(* PLC project Hello Mixing tank, CODESYS CODESYS V3.5 SP16, author Toni Kucic *)
(* stored: creationDateTime 2021-03-11T21:02:17.1386427, version 1.0, modificationDateTime 2021-03-11T20:32:57.2894189, organization Tk Automation *)
(* In industrial automation the "hello world" program is a mixing tank. As a part of my portfolio I have written a simple mixing tank controller and a simulator. The project is meant for begginers and for educational purposes. It is published under MIT license. Written in CODESYS 3.5 and in structured text language.

The project is designed in a way that the user can disable the main program and replace it with his own implementation. Simulator and the HMI sees only the IO and HMI global variables so if the user wishes to create an own implementation those variables should be written. On the simulator side the operator can see if the implementation is working correctly. *)

(* values of MODES: MANUAL: System is in manual mode (Operator control); AUTO: System is in auto mode (PLC in control) *)

{attribute 'qualified_only'}
{attribute 'strict'}
TYPE MODES : (MANUAL := 0, AUTO := 1);
END_TYPE

(* values of AUTO_SEQUENCE: DRAINING: Draining state when system is in auto mode; FILLING: Filling state when system is in auto mode; MIXING: Mixing state when system is in auto mode *)

{attribute 'qualified_only'}
{attribute 'strict'}
TYPE AUTO_SEQUENCE : (DRAINING := 0, FILLING := 1, MIXING := 2);
END_TYPE

FUNCTION_BLOCK GenericBistableDeviceModel
  VAR_INPUT
    ActivateCmd : BOOL;  (* Command to activate the device *)
    DeactivateCmd : BOOL;  (* Command to deactivate the device *)
    cfgActTime : TIME := TIME#1s0ms;  (* Time needed to activate the device *)
    cfgDeactTime : TIME := TIME#1s0ms;  (* Time needed to deactivate the device *)
    simActFail : BOOL;  (* Simulates activation fail. If deactivated and activate command true. *)
    simDeactFail : BOOL;  (* Simulates deactivation fail. If activated and deactivate command true. *)
  END_VAR
  VAR_OUTPUT
    Activated : BOOL;  (* TRUE: Device is activated *)
    Deactivated : BOOL;  (* TRUE: Device is deactivated *)
  END_VAR
  VAR
    TransitionDelay : TON;  (* Timer for delaying the commands to change state *)
    vState : USINT := 0;  (* State tracking variable *)
    vStateOld : USINT := 3;  (* Memory of previous state *)
  END_VAR

            CASE vState OF
	0: (*Deactivated*)
		(*On entry do:*)
		IF vState <> vStateOld THEN
			(*Reset timer*)
			TransitionDelay(IN:=FALSE);
			vStateOld := vState;
		END_IF
		TransitionDelay(IN:=ActivateCmd AND NOT simActFail, PT:=cfgActTime);
		IF TransitionDelay.Q THEN
			vState := 1;
		END_IF
	1: (*Activated*)
		(*On entry do:*)
		IF vState <> vStateOld THEN
			(*Reset timer*)
			TransitionDelay(IN:=FALSE);
			vStateOld := vState;
		END_IF
		TransitionDelay(IN:=DeactivateCmd AND NOT simDeactFail, PT:=cfgDeactTime);
		IF TransitionDelay.Q THEN
			vState := 0;
		END_IF
END_CASE
Activated := vState = 1;
Deactivated := vState = 0;
          
END_FUNCTION_BLOCK

PROGRAM simulator
  VAR
    vTankLevel : REAL := 25;  (* Simulated tank level, intialized to 25% *)
    MixerMotor : GenericBistableDeviceModel;  (* Simulated mixer motor *)
    MediumValve1 : GenericBistableDeviceModel;  (* Simulated valve that fills medium 1 *)
    MediumValve2 : GenericBistableDeviceModel;  (* Simulated valve that fills medium 2 *)
    DrainValve : GenericBistableDeviceModel;  (* Simulated valve that drains the tank *)
    vMotorRotating : REAL;  (* Motor activated for HMI *)
  END_VAR

                    (*Motor and valve simulation*)
MixerMotor(
	ActivateCmd := IO.xDO_M1_MixerMotorRunCmd,
	DeactivateCmd := NOT IO.xDO_M1_MixerMotorRunCmd,
	cfgActTime := T#2S,
	cfgDeactTime := T#0S,
	Activated => IO.xDI_M1_MixerMotorRunning);

MediumValve1(
	ActivateCmd := IO.xDO_VV01_Medium1_OpenCmd,
	DeactivateCmd := NOT IO.xDO_VV01_Medium1_OpenCmd,
	cfgActTime := T#1S,
	cfgDeactTime := T#1S,
	Activated => IO.xDI_VV01_Medium1_Opened);

MediumValve2(
	ActivateCmd := IO.xDO_VV02_Medium2_OpenCmd,
	DeactivateCmd := NOT IO.xDO_VV02_Medium2_OpenCmd,
	cfgActTime := T#1S,
	cfgDeactTime := T#1S,
	Activated => IO.xDI_VV02_Medium2_Opened);

DrainValve(
	ActivateCmd := IO.xDO_VV03_TankDrain_OpenCmd,
	DeactivateCmd := NOT IO.xDO_VV03_TankDrain_OpenCmd,
	cfgActTime := T#1S,
	cfgDeactTime := T#1S,
	Activated => IO.xDI_VV03_TankDrain_Opened);
	
(*Tank filling simulation*)
(*Tank fills if either filling valves are open and drains if the drain is open,
if the program overfills it, the tank spills to the spill way*)
vTankLevel :=  vTankLevel
			 + 0.1 * BOOL_TO_REAL(MediumValve1.Activated)
			 + 0.1 * BOOL_TO_REAL(MediumValve2.Activated)
			 - 0.2 * BOOL_TO_REAL(DrainValve.Activated);
vTankLevel := LIMIT(0, vTankLevel, 100);

(*Limit switch simulation*)
IO.xDI_LS01_TankLevelFull := vTankLevel >= 85;
IO.xDI_LS02_TankLevelEmpty := vTankLevel <= 5;

(*HMI *)
vMotorRotating := vMotorRotating + 1 * BOOL_TO_REAL(MixerMotor.Activated);
IF vMotorRotating >= 360 THEN vMotorRotating := 0; END_IF

                  
END_PROGRAM

PROGRAM main
  VAR
    vMode : MODES;  (* Variable to keep track of system mode Manual/Auto *)
    vModeOld : MODES;  (* Memory of last mode *)
    vAutoState : AUTO_SEQUENCE;  (* Variable to track the automatic sequence *)
    MixingTimer : TON;  (* Timer to control the mixing duration *)
  END_VAR

                    (*Functional description:
There are two ways of operation:
	- Manual
	- Automatic
Manual:
	- Operator is able to operate each valve manually
	- Operator is able to operate the mixer motor manually
	- Overfill protections are disabled
	- Operator is able to put the system to auto
	
Automatic:
	- Program will automatically control the valves and the mixing motor if system is in auto
	- If the tanks level is undefined it assumes draining state
	- In draining state, drains the tank until LS02 activates (tank is empty)
	- When tank is empty, it activates the medium 1 and 2 valves, closes the drain valve and the tank is filling up
	- Filling state is until LS01 is activated (Tank is full)
	- Then the mixer motor is mixing for 10 seconds
	- After mixing is completed, drain the whole contents
	- Repeats as long as auto is activated
	
HMI Requirements:
	- Manual / Auto needs to be correctly controlled and displayed
	- If manual, clicking on devices activates or stops them
	- If auto, clicking is not doing anything
	- If auto, system is counting number of cycles completed
	- Devices must clearly display if they are activated or deactivated*)

(*Enabling operator to select auto or manual mode*)
CASE vMode OF
	MODES.AUTO:
		IF HMI.SetToManual THEN
			vMode := Modes.MANUAL;
			HMI.SetToManual := FALSE;
		END_IF
		
	MODES.MANUAL:
		IF HMI.SetToAuto THEN
			vMode := Modes.AUTO;
			HMI.SetToAuto := FALSE;
		END_IF
END_CASE

(*Control of the system*)
CASE vMode OF
	MODES.MANUAL: (*Manual*)
		(*On entry do:*)
		IF vMode <> vModeOld THEN
			vAutoState := AUTO_SEQUENCE.DRAINING;
			vModeOld := vMode;
		END_IF
		
		(*In manual, HMI commands are connected to the IO for starting and stopping the devices*)
		(*Commands are implemented with a latch*)
		IO.xDO_M1_MixerMotorRunCmd := (HMI.MixerRunCmd OR IO.xDI_M1_MixerMotorRunning) AND NOT (HMI.MixerStopCmd);
		IO.xDO_VV01_Medium1_OpenCmd := (HMI.Medium1OpenCmd OR IO.xDI_VV01_Medium1_Opened) AND NOT (HMI.Medium1CloseCmd);
		IO.xDO_VV02_Medium2_OpenCmd := (HMI.Medium2OpenCmd OR IO.xDI_VV02_Medium2_Opened) AND NOT (HMI.Medium2CloseCmd);
		IO.xDO_VV03_TankDrain_OpenCmd := (HMI.DrainOpenCmd OR IO.xDI_VV03_TankDrain_Opened) AND NOT (HMI.DrainCloseCmd);
	
	MODES.AUTO: (*Automatic*)
		(*On entry do:*)
		IF vMode <> vModeOld THEN
			vAutoState := AUTO_SEQUENCE.DRAINING;
			vModeOld := vMode;
		END_IF
		CASE vAutoState OF
			AUTO_SEQUENCE.FILLING:
				(*Make sure other devices are not working*)
				IO.xDO_M1_MixerMotorRunCmd := FALSE;
				IO.xDO_VV03_TankDrain_OpenCmd := FALSE;
				
				(*Open both medium valves and start filling the tank*)
				IO.xDO_VV01_Medium1_OpenCmd := NOT IO.xDI_LS01_TankLevelFull;
				IO.xDO_VV02_Medium2_OpenCmd := NOT IO.xDI_LS01_TankLevelFull;
				
				(*When tank is full, wait for the filling valves to close and then go to mixing state*)
				IF IO.xDI_LS01_TankLevelFull AND NOT (IO.xDI_VV01_Medium1_Opened OR IO.xDI_VV02_Medium2_Opened) THEN
					vAutoState := AUTO_SEQUENCE.MIXING;
				END_IF
			AUTO_SEQUENCE.MIXING:
				(*Make sure other devices are not working*)
				IO.xDO_VV01_Medium1_OpenCmd := FALSE;
				IO.xDO_VV02_Medium2_OpenCmd := FALSE;
				IO.xDO_VV03_TankDrain_OpenCmd := FALSE;
				
				(*Start the mixer motor and mix for 10s*)
				IO.xDO_M1_MixerMotorRunCmd := TRUE;
				MixingTimer(IN:=IO.xDI_M1_MixerMotorRunning, PT:=T#10S);
				
				(*When timer has elapsed 10s, wait for motor to stop running, then go to draining*)
				IF MixingTimer.Q THEN
					IO.xDO_M1_MixerMotorRunCmd := FALSE;
					vAutoState := AUTO_SEQUENCE.DRAINING;
				END_IF
				
			AUTO_SEQUENCE.DRAINING:
				(*Make sure other devices are not working*)
				IO.xDO_M1_MixerMotorRunCmd := FALSE;
				IO.xDO_VV01_Medium1_OpenCmd := FALSE;
				IO.xDO_VV02_Medium2_OpenCmd := FALSE;
				
				(*Open the drain valve and start draining the tank*)
				IO.xDO_VV03_TankDrain_OpenCmd := NOT IO.xDI_LS02_TankLevelEmpty;
				
				(*When the tank is empty, wait for the drain valve to close,then go to filling*)
				IF IO.xDI_LS02_TankLevelEmpty AND NOT IO.xDI_VV03_TankDrain_Opened THEN
					vAutoState := AUTO_SEQUENCE.FILLING;
					HMI.CyclesCompleted := HMI.CyclesCompleted + 1;
				END_IF
		END_CASE
END_CASE

(*Command sanity reset*)
IF IO.xDI_M1_MixerMotorRunning THEN
	HMI.MixerRunCmd := FALSE;
ELSE
	HMI.MixerStopCmd := FALSE;
END_IF
IF IO.xDI_VV01_Medium1_Opened THEN
	HMI.Medium1OpenCmd := FALSE;
ELSE
	HMI.Medium1CloseCmd := FALSE;
END_IF
IF IO.xDI_VV02_Medium2_Opened THEN
	HMI.Medium2OpenCmd := FALSE;
ELSE
	HMI.Medium2CloseCmd := FALSE;
END_IF
IF IO.xDI_VV03_TankDrain_Opened THEN
	HMI.DrainOpenCmd := FALSE;
ELSE
	HMI.DrainCloseCmd := FALSE;
END_IF

(*HMI *)
HMI.MotorRotating := HMI.MotorRotating + 2 * BOOL_TO_REAL(IO.xDI_M1_MixerMotorRunning);
IF HMI.MotorRotating >= 360 THEN HMI.MotorRotating := 0; END_IF
HMI.InAuto := vMode = MODES.AUTO;
HMI.InManual := vMode = MODES.MANUAL;
                  
END_PROGRAM

CONFIGURATION SoftPLC
  RESOURCE Application ON PLC
    {attribute 'qualified_only'}
    VAR_GLOBAL  (* IO *)
      xDI_LS01_TankLevelFull : BOOL;  (* Tank level switch (HIGH) active *)
      xDI_LS02_TankLevelEmpty : BOOL;  (* Tank level switch (LOW) active *)
      xDI_VV01_Medium1_Opened : BOOL;  (* Medium 1 filling valve open *)
      xDI_VV02_Medium2_Opened : BOOL;  (* Medium 2 filling valve open *)
      xDI_VV03_TankDrain_Opened : BOOL;  (* Tank draining valve open *)
      xDI_M1_MixerMotorRunning : BOOL;  (* Mixer motor running *)
      xDO_VV01_Medium1_OpenCmd : BOOL;  (* Medium 1 filling valve open command *)
      xDO_VV02_Medium2_OpenCmd : BOOL;  (* Medium 2 filling valve open command *)
      xDO_VV03_TankDrain_OpenCmd : BOOL;  (* Tank draining valve open command *)
      xDO_M1_MixerMotorRunCmd : BOOL;  (* Mixer motor run command *)
    END_VAR
    {attribute 'qualified_only'}
    VAR_GLOBAL  (* HMI *)
      MixerRunCmd : BOOL;  (* Command to start the mixer *)
      MixerStopCmd : BOOL;  (* Command to stop the mixer *)
      Medium1OpenCmd : BOOL;  (* Command to open medium 1 valve *)
      Medium1CloseCmd : BOOL;  (* Command to close medium 1 valve *)
      Medium2OpenCmd : BOOL;  (* Command to open medium 2 valve *)
      Medium2CloseCmd : BOOL;  (* Command to close medium 2 valve *)
      DrainOpenCmd : BOOL;  (* Command to open drain valve *)
      DrainCloseCmd : BOOL;  (* Command to close drain valve *)
      SetToAuto : BOOL;  (* Command to set the system to auto mode *)
      SetToManual : BOOL;  (* Command to set the system to manual mode *)
      MotorRotating : REAL;  (* HMI Support variables *)
      InAuto : BOOL;  (* System in AUTO *)
      InManual : BOOL;  (* System in MANUAL *)
      CyclesCompleted : UINT;  (* Cycles completed *)
    END_VAR
    TASK Task(INTERVAL := T#20ms, PRIORITY := 1);
    TASK VISU_TASK(INTERVAL := T#20ms, PRIORITY := 31);
    PROGRAM main WITH Task : main;
    PROGRAM simulator WITH Task : simulator;
    PROGRAM VisuElems.Visu_Prg WITH VISU_TASK : VisuElems.Visu_Prg;
  END_RESOURCE
END_CONFIGURATION
